DATA_BLOCK "Axis_FB_DB"
VAR
  IAI_Axis : Array[1..3] of "IAI_BASE_FB";
END_VAR
BEGIN
END_DATA_BLOCK
